TYPE M2SelectAxisProcessArgs :
STRUCT
	///The axis to select
	axis: M2Axes;
END_STRUCT
END_TYPE

(* stored: Version 1.1.0.1, ProductVersion 3.1.4019.2
   DUT M2SelectAxisProcessArgs: Id {fdde32c7-cd3a-4681-9561-eececc5abc9f} *)
